// TIA Portal V17 export
// export: Created 2024-08-07T21:44:06.3119046Z, ExportSetting WithDefaults, DisplayName Totally Integrated Automation Portal, DisplayVersion V17 Update 7, DisplayName TIA Portal Openness, DisplayVersion V17 Update 7, DisplayName TIA Portal Version Control Interface, DisplayVersion V17, DisplayName SINAMICS Startdrive Advanced, DisplayVersion V17 SP2, DisplayName SINAMICS Startdrive G110M, G120, G120C, G120D, G120P, G115D, DisplayVersion V17 SP2, DisplayName SINAMICS Startdrive G130, G150, S120, S150, SINAMICS MV, S210, DisplayVersion V17 SP2, DisplayName STEP 7 Professional, DisplayVersion V17 Update 7, DisplayName STEP 7 Safety, DisplayVersion V17 Update 6, DisplayName WinCC Advanced / Unified PC, DisplayVersion V17 Update 7
FUNCTION_BLOCK "sq_autoeject"   // FB53, GRAPH
VERSION : 0.1
// stored: AcknowledgeErrorsRequired true, AutoNumber true, GraphVersion 6.0, InitialValuesAcquisition false, IsIECCheckEnabled false, LanguageInNetworks LAD, LockOperatingMode false, PermanentILProcessingInMANMode false, SetENOAutomatically false, SkipSteps false, UDAEnableTagReadback false, WithAlarmHandling true
   // inherited from GRAPH_BASE
   VAR
      OFF_SQ_BASE : Bool;
   END_VAR
   VAR_INPUT
      OFF_SQ { ExternalWritable := 'False'} : Bool := false;   // Turn sequence off
      INIT_SQ { ExternalWritable := 'False'} : Bool := false;   // Set sequence to initial state
      ACK_EF { ExternalWritable := 'False'} : Bool := false;   // Acknowledge all errors and faults
      S_PREV { ExternalWritable := 'False'} : Bool := false;   // Output previous step in parameter S_NO
      S_NEXT { ExternalWritable := 'False'} : Bool := false;   // Indicate next step in parameter S_NO
      SW_AUTO { ExternalWritable := 'False'} : Bool := false;   // Automatic mode
      SW_TAP { ExternalWritable := 'False'} : Bool := false;   // Semiautomatic/switch with transition
      SW_TOP { ExternalWritable := 'False'} : Bool := false;   // Semiautomatic/ignore transition
      SW_MAN { ExternalWritable := 'False'} : Bool := false;   // Manual mode
      S_SEL { ExternalWritable := 'False'} : Int := 0;   // Select step to be output to S_NO
      S_ON { ExternalWritable := 'False'} : Bool := false;   // Activate step indicated in S_NO
      S_OFF { ExternalWritable := 'False'} : Bool := false;   // Deactivate step indicated S_NO
      T_PUSH { ExternalWritable := 'False'} : Bool := false;   // Enable transition to switch in semi automatic mode
   END_VAR
   VAR_OUTPUT
      S_NO { ExternalWritable := 'False'} : Int := 0;   // Step number
      S_MORE { ExternalWritable := 'False'} : Bool := false;   // More steps are available and can be shown in S_NO
      S_ACTIVE { ExternalWritable := 'False'} : Bool := false;   // Step indicated in S_NO is active
      ERR_FLT { ExternalWritable := 'False'} : Bool := false;   // Interlock or supervision group error
      AUTO_ON { ExternalWritable := 'False'} : Bool := false;   // Automatic mode is active
      TAP_ON { ExternalWritable := 'False'} : Bool := false;   // Semiautomatic mode/step with transition enabled
      TOP_ON { ExternalWritable := 'False'} : Bool := false;   // Semiautomatic mode/ignore transition enabled
      MAN_ON { ExternalWritable := 'False'} : Bool := false;   // Manual mode is active
   END_VAR
   VAR
      dummy : Bool;
      start : Bool;
      base : Bool;
   END_VAR
BEGIN
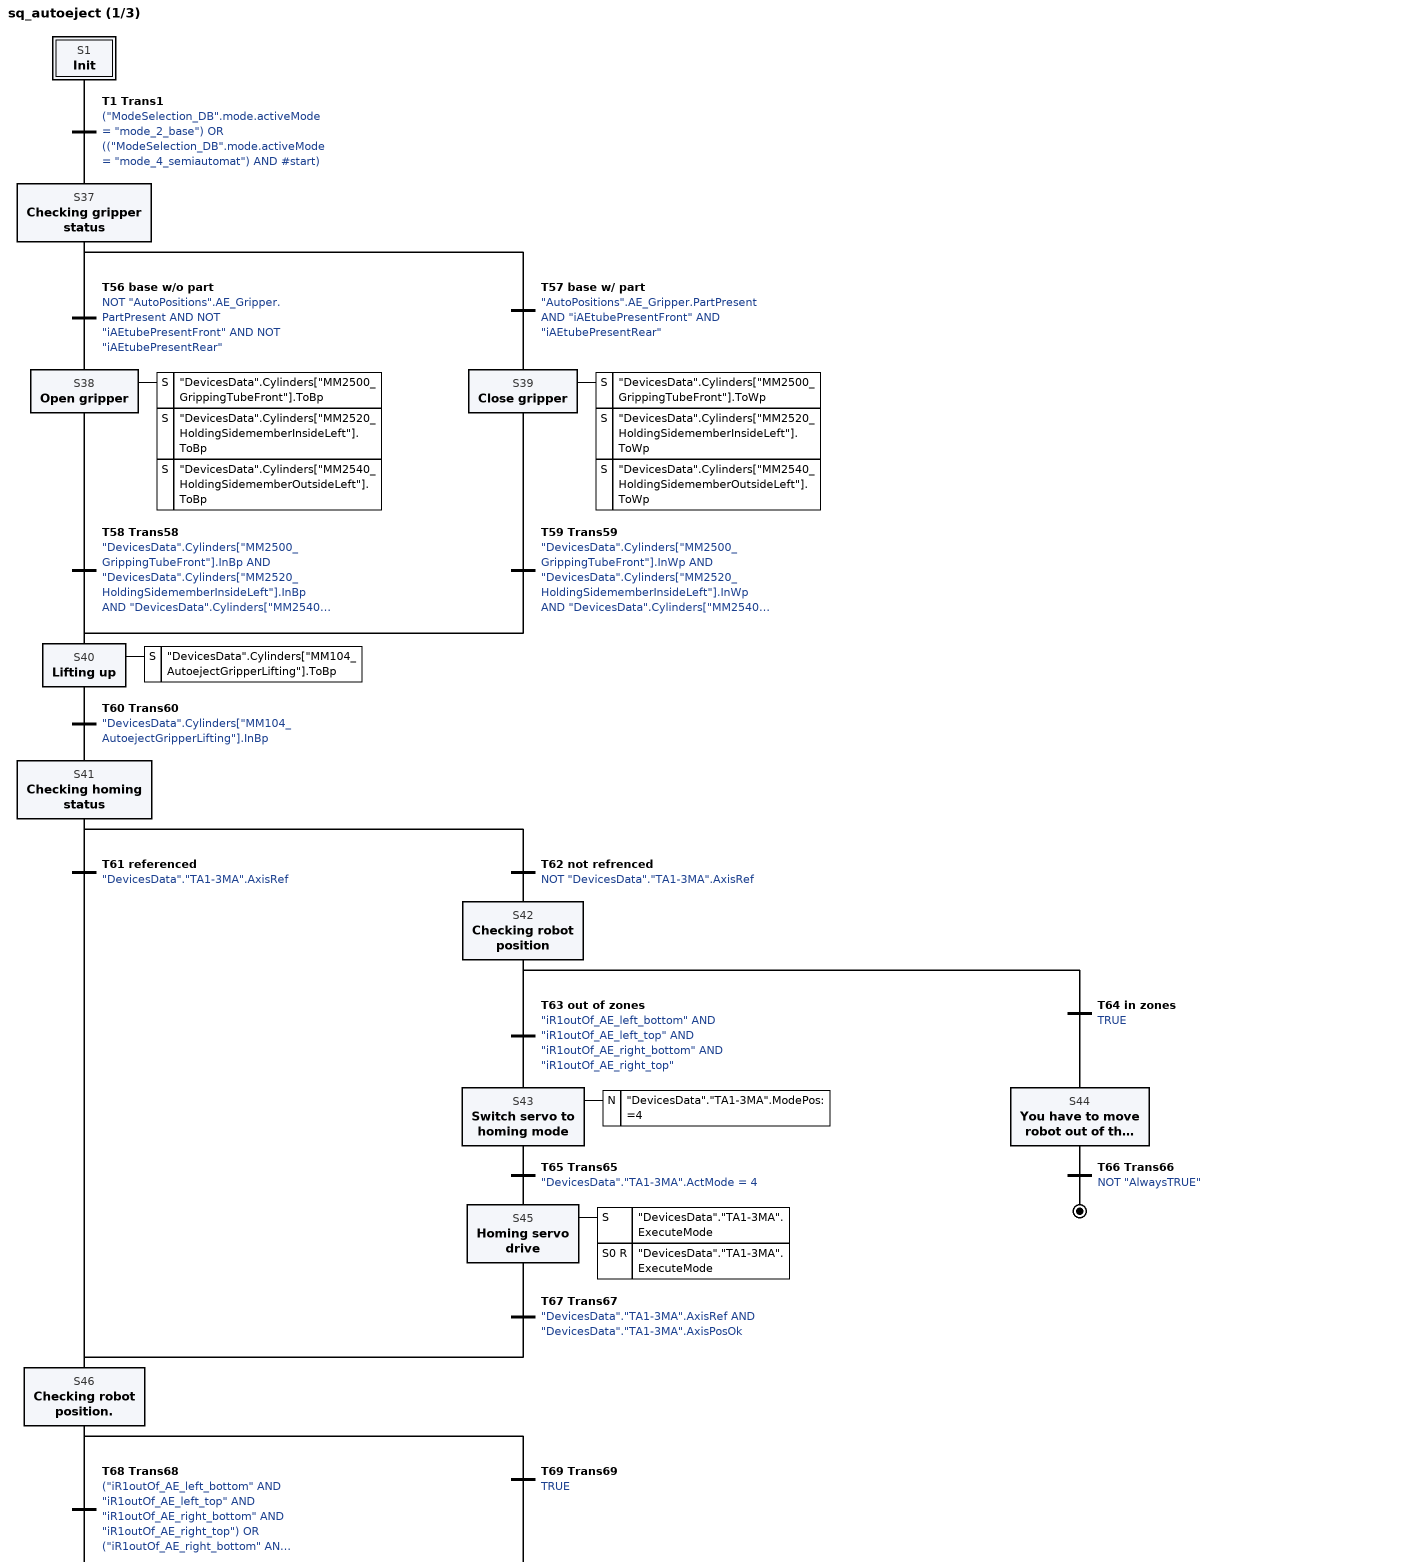
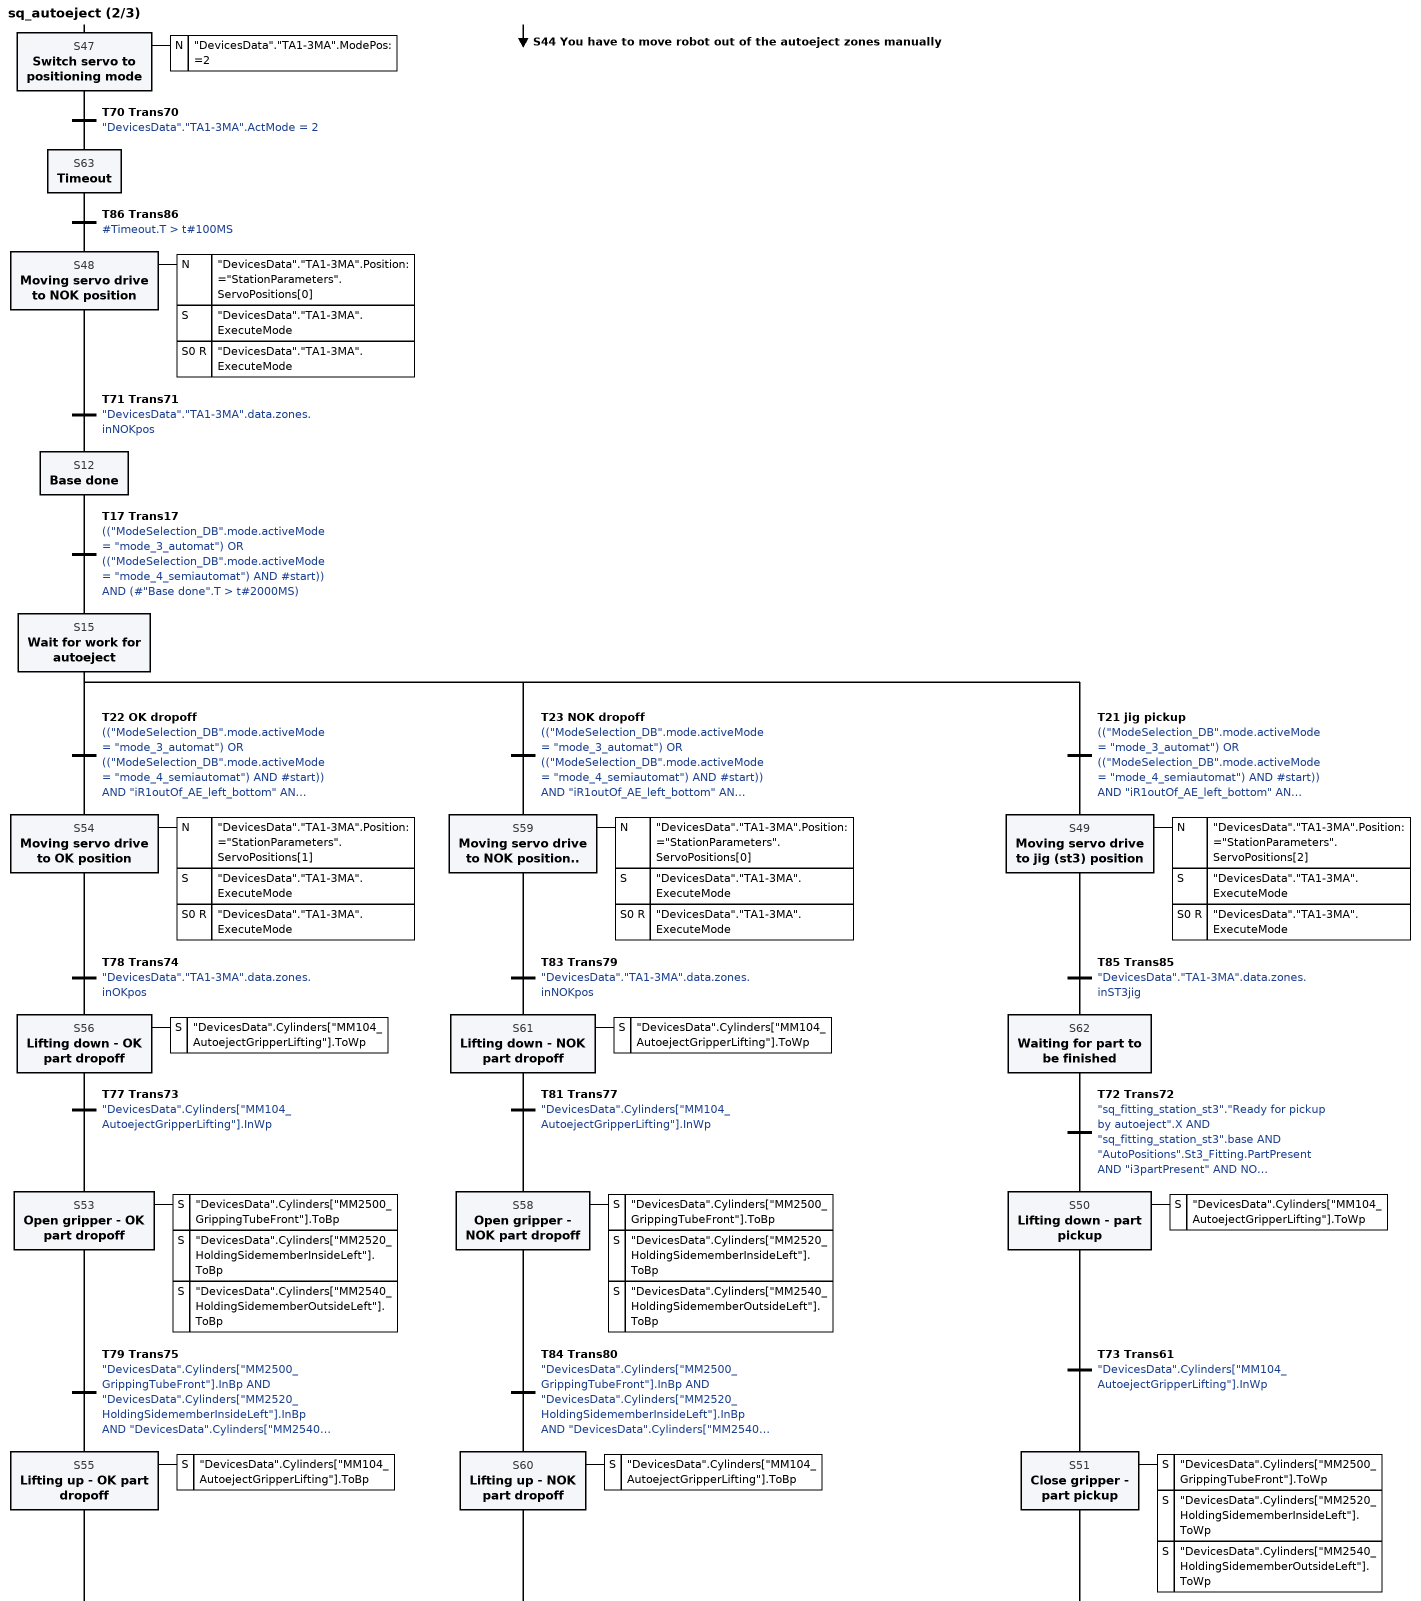
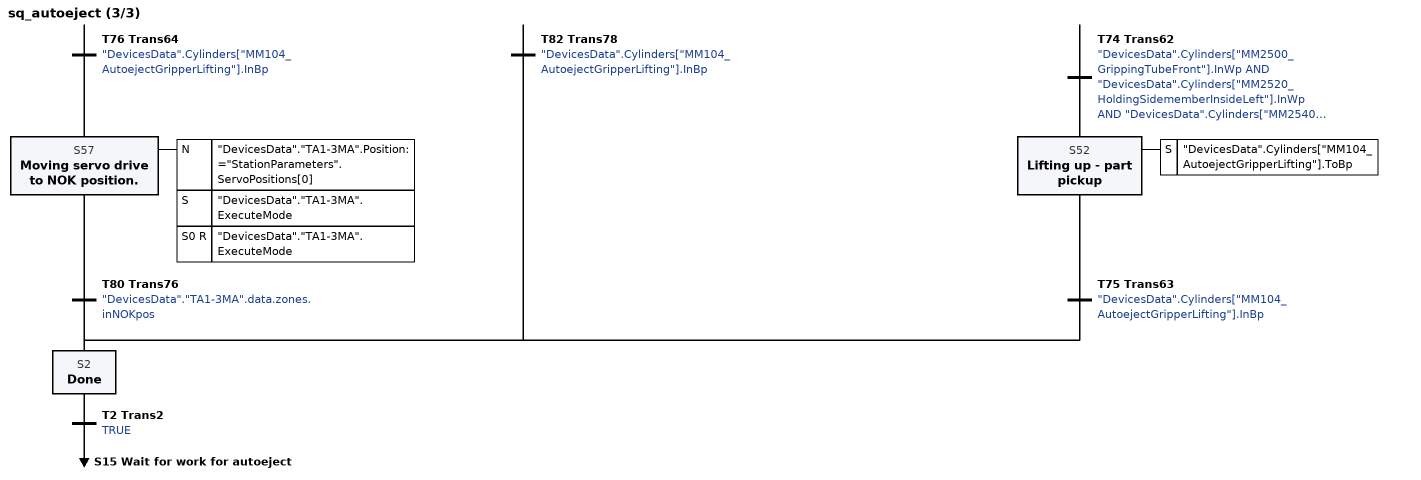
   // sequencer 1
   INITIAL_STEP Init:   // S1, max time T#10S, warning time T#7S
   END_STEP
   TRANSITION Trans1 FROM Init TO "Checking gripper status"   // T1
      := ("ModeSelection_DB".mode.activeMode = "mode_2_base") OR (("ModeSelection_DB".mode.activeMode = "mode_4_semiautomat") AND #start);
   END_TRANSITION
   STEP Done:   // S2, max time T#10S, warning time T#7S
   END_STEP
   TRANSITION Trans2 FROM Done TO "Wait for work for autoeject"   // T2, jump
      := TRUE;
   END_TRANSITION
   STEP "Base done":   // S12, max time T#10S, warning time T#7S
   END_STEP
   TRANSITION Trans17 FROM "Base done" TO "Wait for work for autoeject"   // T17
      := (("ModeSelection_DB".mode.activeMode = "mode_3_automat") OR (("ModeSelection_DB".mode.activeMode = "mode_4_semiautomat") AND #start)) AND (#"Base done".T > t#2000MS);
   END_TRANSITION
   STEP "Wait for work for autoeject":   // S15, max time T#10S, warning time T#7S
   END_STEP
   TRANSITION "OK dropoff" FROM "Wait for work for autoeject" TO "Moving servo drive to OK position"   // T22
      := (("ModeSelection_DB".mode.activeMode = "mode_3_automat") OR (("ModeSelection_DB".mode.activeMode = "mode_4_semiautomat") AND #start)) AND "iR1outOf_AE_left_bottom" AND "iR1outOf_AE_left_top" AND "iR1outOf_AE_right_bottom" AND "iR1outOf_AE_right_top" AND "AutoPositions".AE_Gripper.PartPresent AND "AutoPositions".AE_Gripper.StFinished[3] AND NOT "AutoPositions".AE_Gripper.PartNOK AND "iAEtubePresentFront" AND "iAEtubePresentRear" AND NOT "AutoPositions".St4_OKposition.PartPresent AND NOT "i4partPresent";
   END_TRANSITION
   TRANSITION "NOK dropoff" FROM "Wait for work for autoeject" TO "Moving servo drive to NOK position.."   // T23
      := (("ModeSelection_DB".mode.activeMode = "mode_3_automat") OR (("ModeSelection_DB".mode.activeMode = "mode_4_semiautomat") AND #start)) AND "iR1outOf_AE_left_bottom" AND "iR1outOf_AE_left_top" AND "iR1outOf_AE_right_bottom" AND "iR1outOf_AE_right_top" AND "AutoPositions".AE_Gripper.PartPresent AND (NOT "AutoPositions".AE_Gripper.StFinished[3] OR "AutoPositions".AE_Gripper.PartNOK) AND "iAEtubePresentFront" AND "iAEtubePresentRear" AND NOT "PartHolderData".NOKBoxFull;
   END_TRANSITION
   TRANSITION "jig pickup" FROM "Wait for work for autoeject" TO "Moving servo drive to jig (st3) position"   // T21
      := (("ModeSelection_DB".mode.activeMode = "mode_3_automat") OR (("ModeSelection_DB".mode.activeMode = "mode_4_semiautomat") AND #start)) AND "iR1outOf_AE_left_bottom" AND "iR1outOf_AE_left_top" AND "iR1outOf_AE_right_bottom" AND "iR1outOf_AE_right_top" AND "AutoPositions".St3_Fitting.PartPresent AND "i3partPresent" AND NOT "AutoPositions".AE_Gripper.PartPresent AND NOT "iAEtubePresentFront" AND NOT "iAEtubePresentRear" AND NOT "AutoPositions".St4_OKposition.PartPresent AND NOT "i4partPresent";
   END_TRANSITION
   STEP "Close gripper - part pickup":   // S51, max time T#10S, warning time T#7S
              S    "DevicesData".Cylinders["MM2500_GrippingTubeFront"].ToWp
              S    "DevicesData".Cylinders["MM2520_HoldingSidememberInsideLeft"].ToWp
              S    "DevicesData".Cylinders["MM2540_HoldingSidememberOutsideLeft"].ToWp
   END_STEP
   TRANSITION Trans62 FROM "Close gripper - part pickup" TO "Lifting up - part pickup"   // T74
      := "DevicesData".Cylinders["MM2500_GrippingTubeFront"].InWp AND "DevicesData".Cylinders["MM2520_HoldingSidememberInsideLeft"].InWp AND "DevicesData".Cylinders["MM2540_HoldingSidememberOutsideLeft"].InWp;
   END_TRANSITION
   STEP "Open gripper - OK part dropoff":   // S53, max time T#10S, warning time T#7S
              S    "DevicesData".Cylinders["MM2500_GrippingTubeFront"].ToBp
              S    "DevicesData".Cylinders["MM2520_HoldingSidememberInsideLeft"].ToBp
              S    "DevicesData".Cylinders["MM2540_HoldingSidememberOutsideLeft"].ToBp
   END_STEP
   TRANSITION Trans75 FROM "Open gripper - OK part dropoff" TO "Lifting up - OK part dropoff"   // T79
      := "DevicesData".Cylinders["MM2500_GrippingTubeFront"].InBp AND "DevicesData".Cylinders["MM2520_HoldingSidememberInsideLeft"].InBp AND "DevicesData".Cylinders["MM2540_HoldingSidememberOutsideLeft"].InBp;
   END_TRANSITION
   STEP "Moving servo drive to OK position":   // S54, max time T#30S, warning time T#7S
      supervision V := #"Moving servo drive to OK position".T > #"Moving servo drive to OK position".T_MAX;
              N    "DevicesData"."TA1-3MA".Position:="StationParameters".ServoPositions[1]
              S    "DevicesData"."TA1-3MA".ExecuteMode
          S0  R    "DevicesData"."TA1-3MA".ExecuteMode
   END_STEP
   TRANSITION Trans74 FROM "Moving servo drive to OK position" TO "Lifting down - OK part dropoff"   // T78
      := "DevicesData"."TA1-3MA".data.zones.inOKpos;
   END_TRANSITION
   STEP "Lifting up - OK part dropoff":   // S55, max time T#10S, warning time T#7S
              S    "DevicesData".Cylinders["MM104_AutoejectGripperLifting"].ToBp
   END_STEP
   TRANSITION Trans64 FROM "Lifting up - OK part dropoff" TO "Moving servo drive to NOK position."   // T76
      := "DevicesData".Cylinders["MM104_AutoejectGripperLifting"].InBp;
   END_TRANSITION
   STEP "Lifting down - OK part dropoff":   // S56, max time T#10S, warning time T#7S
              S    "DevicesData".Cylinders["MM104_AutoejectGripperLifting"].ToWp
   END_STEP
   TRANSITION Trans73 FROM "Lifting down - OK part dropoff" TO "Open gripper - OK part dropoff"   // T77
      := "DevicesData".Cylinders["MM104_AutoejectGripperLifting"].InWp;
   END_TRANSITION
   STEP "Moving servo drive to jig (st3) position":   // S49, max time T#30S, warning time T#7S
      supervision V := #"Moving servo drive to jig (st3) position".T > #"Moving servo drive to jig (st3) position".T_MAX;
              N    "DevicesData"."TA1-3MA".Position:="StationParameters".ServoPositions[2]
              S    "DevicesData"."TA1-3MA".ExecuteMode
          S0  R    "DevicesData"."TA1-3MA".ExecuteMode
   END_STEP
   TRANSITION Trans85 FROM "Moving servo drive to jig (st3) position" TO "Waiting for part to be finished"   // T85
      := "DevicesData"."TA1-3MA".data.zones.inST3jig;
   END_TRANSITION
   STEP "Lifting up - part pickup":   // S52, max time T#10S, warning time T#7S
              S    "DevicesData".Cylinders["MM104_AutoejectGripperLifting"].ToBp
   END_STEP
   TRANSITION Trans63 FROM "Lifting up - part pickup" TO Done   // T75
      := "DevicesData".Cylinders["MM104_AutoejectGripperLifting"].InBp;
   END_TRANSITION
   STEP "Lifting down - part pickup":   // S50, max time T#10S, warning time T#7S
              S    "DevicesData".Cylinders["MM104_AutoejectGripperLifting"].ToWp
   END_STEP
   TRANSITION Trans61 FROM "Lifting down - part pickup" TO "Close gripper - part pickup"   // T73
      := "DevicesData".Cylinders["MM104_AutoejectGripperLifting"].InWp;
   END_TRANSITION
   STEP "Checking gripper status":   // S37, max time T#10S, warning time T#7S
   END_STEP
   TRANSITION "base w/o part" FROM "Checking gripper status" TO "Open gripper"   // T56
      := NOT "AutoPositions".AE_Gripper.PartPresent AND NOT "iAEtubePresentFront" AND NOT "iAEtubePresentRear";
   END_TRANSITION
   TRANSITION "base w/ part" FROM "Checking gripper status" TO "Close gripper"   // T57
      := "AutoPositions".AE_Gripper.PartPresent AND "iAEtubePresentFront" AND "iAEtubePresentRear";
   END_TRANSITION
   STEP "Open gripper":   // S38, max time T#10S, warning time T#7S
              S    "DevicesData".Cylinders["MM2500_GrippingTubeFront"].ToBp
              S    "DevicesData".Cylinders["MM2520_HoldingSidememberInsideLeft"].ToBp
              S    "DevicesData".Cylinders["MM2540_HoldingSidememberOutsideLeft"].ToBp
   END_STEP
   TRANSITION Trans58 FROM "Open gripper" TO "Lifting up"   // T58
      := "DevicesData".Cylinders["MM2500_GrippingTubeFront"].InBp AND "DevicesData".Cylinders["MM2520_HoldingSidememberInsideLeft"].InBp AND "DevicesData".Cylinders["MM2540_HoldingSidememberOutsideLeft"].InBp;
   END_TRANSITION
   STEP "Close gripper":   // S39, max time T#10S, warning time T#7S
              S    "DevicesData".Cylinders["MM2500_GrippingTubeFront"].ToWp
              S    "DevicesData".Cylinders["MM2520_HoldingSidememberInsideLeft"].ToWp
              S    "DevicesData".Cylinders["MM2540_HoldingSidememberOutsideLeft"].ToWp
   END_STEP
   TRANSITION Trans59 FROM "Close gripper" TO "Lifting up"   // T59
      := "DevicesData".Cylinders["MM2500_GrippingTubeFront"].InWp AND "DevicesData".Cylinders["MM2520_HoldingSidememberInsideLeft"].InWp AND "DevicesData".Cylinders["MM2540_HoldingSidememberOutsideLeft"].InWp;
   END_TRANSITION
   STEP "Lifting up":   // S40, max time T#10S, warning time T#7S
              S    "DevicesData".Cylinders["MM104_AutoejectGripperLifting"].ToBp
   END_STEP
   TRANSITION Trans60 FROM "Lifting up" TO "Checking homing status"   // T60
      := "DevicesData".Cylinders["MM104_AutoejectGripperLifting"].InBp;
   END_TRANSITION
   STEP "Checking homing status":   // S41, max time T#10S, warning time T#7S
   END_STEP
   TRANSITION referenced FROM "Checking homing status" TO "Checking robot position."   // T61
      := "DevicesData"."TA1-3MA".AxisRef;
   END_TRANSITION
   TRANSITION "not refrenced" FROM "Checking homing status" TO "Checking robot position"   // T62
      := NOT "DevicesData"."TA1-3MA".AxisRef;
   END_TRANSITION
   STEP "Checking robot position":   // S42, max time T#10S, warning time T#7S
   END_STEP
   TRANSITION "out of zones" FROM "Checking robot position" TO "Switch servo to homing mode"   // T63
      := "iR1outOf_AE_left_bottom" AND "iR1outOf_AE_left_top" AND "iR1outOf_AE_right_bottom" AND "iR1outOf_AE_right_top";
   END_TRANSITION
   TRANSITION "in zones" FROM "Checking robot position" TO "You have to move robot out of the autoeject zones manually"   // T64
      := TRUE;
   END_TRANSITION
   STEP "Switch servo to homing mode":   // S43, max time T#10S, warning time T#7S
      supervision V := #"Switch servo to homing mode".T > #"Switch servo to homing mode".T_MAX;
              N    "DevicesData"."TA1-3MA".ModePos:=4
   END_STEP
   TRANSITION Trans65 FROM "Switch servo to homing mode" TO "Homing servo drive"   // T65
      := "DevicesData"."TA1-3MA".ActMode = 4;
   END_TRANSITION
   STEP "You have to move robot out of the autoeject zones manually":   // S44, max time T#10S, warning time T#7S
      supervision V := "AlwaysTRUE";
   END_STEP
   TRANSITION Trans66 FROM "You have to move robot out of the autoeject zones manually" TO END   // T66
      := NOT "AlwaysTRUE";
   END_TRANSITION
   STEP "Homing servo drive":   // S45, max time T#30S, warning time T#7S
      supervision V := #"Homing servo drive".T > #"Homing servo drive".T_MAX;
              S    "DevicesData"."TA1-3MA".ExecuteMode
          S0  R    "DevicesData"."TA1-3MA".ExecuteMode
   END_STEP
   TRANSITION Trans67 FROM "Homing servo drive" TO "Checking robot position."   // T67
      := "DevicesData"."TA1-3MA".AxisRef AND "DevicesData"."TA1-3MA".AxisPosOk;
   END_TRANSITION
   STEP "Checking robot position.":   // S46, max time T#10S, warning time T#7S
   END_STEP
   TRANSITION Trans68 FROM "Checking robot position." TO "Switch servo to positioning mode"   // T68
      := ("iR1outOf_AE_left_bottom" AND "iR1outOf_AE_left_top" AND "iR1outOf_AE_right_bottom" AND "iR1outOf_AE_right_top") OR ("iR1outOf_AE_right_bottom" AND "iR1outOf_AE_right_top" AND "DevicesData"."TA1-3MA".data.zones.outOfST3zone);
   END_TRANSITION
   TRANSITION Trans69 FROM "Checking robot position." TO "You have to move robot out of the autoeject zones manually"   // T69, jump
      := TRUE;
   END_TRANSITION
   STEP "Switch servo to positioning mode":   // S47, max time T#10S, warning time T#7S
      supervision V := #"Switch servo to positioning mode".T > #"Switch servo to positioning mode".T_MAX;
              N    "DevicesData"."TA1-3MA".ModePos:=2
   END_STEP
   TRANSITION Trans70 FROM "Switch servo to positioning mode" TO Timeout   // T70
      := "DevicesData"."TA1-3MA".ActMode = 2;
   END_TRANSITION
   STEP "Moving servo drive to NOK position":   // S48, max time T#30S, warning time T#7S
      supervision V := #"Moving servo drive to NOK position".T > #"Moving servo drive to NOK position".T_MAX;
              N    "DevicesData"."TA1-3MA".Position:="StationParameters".ServoPositions[0]
              S    "DevicesData"."TA1-3MA".ExecuteMode
          S0  R    "DevicesData"."TA1-3MA".ExecuteMode
   END_STEP
   TRANSITION Trans71 FROM "Moving servo drive to NOK position" TO "Base done"   // T71
      := "DevicesData"."TA1-3MA".data.zones.inNOKpos;
   END_TRANSITION
   STEP "Moving servo drive to NOK position.":   // S57, max time T#30S, warning time T#7S
      supervision V := #"Moving servo drive to NOK position.".T > #"Moving servo drive to NOK position.".T_MAX;
              N    "DevicesData"."TA1-3MA".Position:="StationParameters".ServoPositions[0]
              S    "DevicesData"."TA1-3MA".ExecuteMode
          S0  R    "DevicesData"."TA1-3MA".ExecuteMode
   END_STEP
   TRANSITION Trans76 FROM "Moving servo drive to NOK position." TO Done   // T80
      := "DevicesData"."TA1-3MA".data.zones.inNOKpos;
   END_TRANSITION
   STEP "Open gripper - NOK part dropoff":   // S58, max time T#10S, warning time T#7S
              S    "DevicesData".Cylinders["MM2500_GrippingTubeFront"].ToBp
              S    "DevicesData".Cylinders["MM2520_HoldingSidememberInsideLeft"].ToBp
              S    "DevicesData".Cylinders["MM2540_HoldingSidememberOutsideLeft"].ToBp
   END_STEP
   TRANSITION Trans80 FROM "Open gripper - NOK part dropoff" TO "Lifting up - NOK part dropoff"   // T84
      := "DevicesData".Cylinders["MM2500_GrippingTubeFront"].InBp AND "DevicesData".Cylinders["MM2520_HoldingSidememberInsideLeft"].InBp AND "DevicesData".Cylinders["MM2540_HoldingSidememberOutsideLeft"].InBp;
   END_TRANSITION
   STEP "Moving servo drive to NOK position..":   // S59, max time T#30S, warning time T#7S
      supervision V := #"Moving servo drive to NOK position..".T > #"Moving servo drive to NOK position..".T_MAX;
              N    "DevicesData"."TA1-3MA".Position:="StationParameters".ServoPositions[0]
              S    "DevicesData"."TA1-3MA".ExecuteMode
          S0  R    "DevicesData"."TA1-3MA".ExecuteMode
   END_STEP
   TRANSITION Trans79 FROM "Moving servo drive to NOK position.." TO "Lifting down - NOK part dropoff"   // T83
      := "DevicesData"."TA1-3MA".data.zones.inNOKpos;
   END_TRANSITION
   STEP "Lifting up - NOK part dropoff":   // S60, max time T#10S, warning time T#7S
              S    "DevicesData".Cylinders["MM104_AutoejectGripperLifting"].ToBp
   END_STEP
   TRANSITION Trans78 FROM "Lifting up - NOK part dropoff" TO Done   // T82
      := "DevicesData".Cylinders["MM104_AutoejectGripperLifting"].InBp;
   END_TRANSITION
   STEP "Lifting down - NOK part dropoff":   // S61, max time T#10S, warning time T#7S
              S    "DevicesData".Cylinders["MM104_AutoejectGripperLifting"].ToWp
   END_STEP
   TRANSITION Trans77 FROM "Lifting down - NOK part dropoff" TO "Open gripper - NOK part dropoff"   // T81
      := "DevicesData".Cylinders["MM104_AutoejectGripperLifting"].InWp;
   END_TRANSITION
   STEP "Waiting for part to be finished":   // S62, max time T#10S, warning time T#7S
   END_STEP
   TRANSITION Trans72 FROM "Waiting for part to be finished" TO "Lifting down - part pickup"   // T72
      := "sq_fitting_station_st3"."Ready for pickup by autoeject".X AND "sq_fitting_station_st3".base AND "AutoPositions".St3_Fitting.PartPresent AND "i3partPresent" AND NOT "AutoPositions".AE_Gripper.PartPresent AND NOT "iAEtubePresentFront" AND NOT "iAEtubePresentRear" AND NOT "AutoPositions".St4_OKposition.PartPresent;
   END_TRANSITION
   STEP Timeout:   // S63, max time T#10S, warning time T#7S
   END_STEP
   TRANSITION Trans86 FROM Timeout TO "Moving servo drive to NOK position"   // T86
      := #Timeout.T > t#100MS;
   END_TRANSITION
END_FUNCTION_BLOCK
